// TIA Portal V17 export
// export: Created 2021-12-03T08:08:09.4318727Z, ExportSetting WithDefaults, DisplayName Totally Integrated Automation Portal, DisplayVersion V17, DisplayName TIA Portal Openness, DisplayVersion V17, DisplayName TIA Portal Version Control Interface, DisplayVersion V17, DisplayName STEP 7 Professional, DisplayVersion V17, DisplayName STEP 7 Safety, DisplayVersion V17, DisplayName WinCC Advanced, DisplayVersion V17
VAR_GLOBAL   // PLC tag table "Faults"
   CirBrk24VFb AT %MW140 : Int;
   CirBrk24VFb_1 AT %M140.1 : Bool;
   CirBrk24VFb_2 AT %M140.2 : Bool;
   CirBrk24VFb_3 AT %M140.3 : Bool;
   CirBrk24VFb_4 AT %M140.4 : Bool;
   CirBrk24VFb_5 AT %M140.5 : Bool;
   CirBrk24VFb_6 AT %M140.6 : Bool;
   CirBrk24VFb_7 AT %M140.7 : Bool;
   CirBrk24VFb_8 AT %M141.0 : Bool;
   CirBrk24VFb_9 AT %M141.1 : Bool;
   CirBrk24VFb_10 AT %M141.2 : Bool;
   CirBrk24VFb_11 AT %M141.3 : Bool;
   CirBrk24VFb_12 AT %M141.4 : Bool;
   CirBrk24VFb_13 AT %M141.5 : Bool;
   CirBrk24VFb_14 AT %M141.6 : Bool;
   CirBrk24VFb_15 AT %M141.7 : Bool;
   CirBrk220VFb AT %MW142 : Int;
   CirBrk220VFb_1 AT %M142.1 : Bool;
   CirBrk220VFb_2 AT %M142.2 : Bool;
   CirBrk220VFb_3 AT %M142.3 : Bool;
   CirBrk220VFb_4 AT %M142.4 : Bool;
   CirBrk220VFb_5 AT %M142.5 : Bool;
   CirBrk220VFb_6 AT %M142.6 : Bool;
   CirBrk220VFb_7 AT %M142.7 : Bool;
   CirBrk220VFb_8 AT %M143.0 : Bool;
   CirBrk220VFb_9 AT %M143.1 : Bool;
   CirBrk220VFb_10 AT %M143.2 : Bool;
   CirBrk220VFb_11 AT %M143.3 : Bool;
   CirBrk220VFb_12 AT %M143.4 : Bool;
   CirBrk220VFb_13 AT %M143.5 : Bool;
   CirBrk220VFb_14 AT %M143.6 : Bool;
   CirBrk220VFb_15 AT %M143.7 : Bool;
   CirBrk380VFb AT %MW144 : Int;
   CirBrk380VFb_1 AT %M144.1 : Bool;
   CirBrk380VFb_2 AT %M144.2 : Bool;
   CirBrk380VFb_3 AT %M144.3 : Bool;
   CirBrk380VFb_4 AT %M144.4 : Bool;
   CirBrk380VFb_5 AT %M144.5 : Bool;
   CirBrk380VFb_6 AT %M144.6 : Bool;
   CirBrk380VFb_7 AT %M144.7 : Bool;
   CirBrk380VFb_8 AT %M145.0 : Bool;
   CirBrk380VFb_9 AT %M145.1 : Bool;
   CirBrk380VFb_10 AT %M145.2 : Bool;
   CirBrk380VFb_11 AT %M145.3 : Bool;
   CirBrk380VFb_12 AT %M145.4 : Bool;
   CirBrk380VFb_13 AT %M145.5 : Bool;
   CirBrk380VFb_14 AT %M145.6 : Bool;
   CirBrk380VFb_15 AT %M145.7 : Bool;
   FitBackControl AT %MW146 : Int;
   FitBackControl_1 AT %M146.1 : Bool;
   FitBackControl_2 AT %M146.2 : Bool;
   FitBackControl_3 AT %M146.3 : Bool;
   FitBackControl_4 AT %M146.4 : Bool;
   FitBackControl_5 AT %M146.5 : Bool;
   FitBackControl_6 AT %M146.6 : Bool;
   FitBackControl_7 AT %M146.7 : Bool;
   FitBackControl_8 AT %M147.0 : Bool;
   FitBackControl_9 AT %M147.1 : Bool;
   FitBackControl_10 AT %M147.2 : Bool;
   FitBackControl_11 AT %M147.3 : Bool;
   FitBackControl_12 AT %M147.4 : Bool;
   FitBackControl_13 AT %M147.5 : Bool;
   FitBackControl_14 AT %M147.6 : Bool;
   FitBackControl_15 AT %M147.7 : Bool;
   EmStBt AT %MW148 : Int;
   EmStBt_1 AT %M148.1 : Bool;
   EmStBt_2 AT %M148.2 : Bool;
   EmStBt_3 AT %M148.3 : Bool;
   EmStBt_4 AT %M148.4 : Bool;
   EmStBt_5 AT %M148.5 : Bool;
   EmStBt_6 AT %M148.6 : Bool;
   EmStBt_7 AT %M148.7 : Bool;
   EmStBt_8 AT %M149.0 : Bool;
   EmStBt_9 AT %M149.1 : Bool;
   EmStBt_10 AT %M149.2 : Bool;
   EmStBt_11 AT %M149.3 : Bool;
   EmStBt_12 AT %M149.4 : Bool;
   EmStBt_13 AT %M149.5 : Bool;
   EmStBt_14 AT %M149.6 : Bool;
   EmStBt_15 AT %M149.7 : Bool;
   Conveyer AT %MW150 : Int;
   Conveyer_1 AT %M150.1 : Bool;
   Conveyer_2 AT %M150.2 : Bool;
   Conveyer_3 AT %M150.3 : Bool;
   Conveyer_4 AT %M150.4 : Bool;
   Conveyer_5 AT %M150.5 : Bool;
   Conveyer_6 AT %M150.6 : Bool;
   Conveyer_7 AT %M150.7 : Bool;
   Conveyer_8 AT %M151.0 : Bool;
   Conveyer_9 AT %M151.1 : Bool;
   Conveyer_10 AT %M151.2 : Bool;
   Conveyer_11 AT %M151.3 : Bool;
   Conveyer_12 AT %M151.4 : Bool;
   Conveyer_13 AT %M151.5 : Bool;
   Conveyer_14 AT %M151.6 : Bool;
   Conveyer_15 AT %M151.7 : Bool;
   CirBrk24VFb_0 AT %M140.0 : Bool;
   CirBrk220VFb_0 AT %M142.0 : Bool;
   CirBrk380VFb_0 AT %M144.0 : Bool;
   FitBackControl_0 AT %M146.0 : Bool;
   EmStBt_0 AT %M148.0 : Bool;
   Conveyer_0 AT %M150.0 : Bool;
END_VAR
